PROGRAM Main
VAR
	type_test : TypeTest;
	write_test : WriteTest;
	// Struct packing test targets — one instance per pack_mode
	// struct_tests: PLC drives these from seed (Go read-only for phase 1)
	struct_test : StructTest;
	
	{attribute 'some_made_up_var_key':='some_made_up_var_value'}
	attribute_test : AttributeTest;
END_VAR

type_test();
write_test();
struct_test();
attribute_test();

END_PROGRAM

(* stored: Version 1.1.0.1, ProductVersion 3.1.4024.13
   POU Main: Id {151bda18-a213-42d0-86e0-e79837f085e9}, SpecialFunc None *)
